# EPICS autosave request: apps/iocBoot/iocftcTemps/OmegaCYD218_All_settings.req
file "OmegaCYD218_settings.req" P=B_HW_FTC:CYD218_0:
file "OmegaCYD218_settings.req" P=B_HW_FTC:CYD218_1:
